Fanuc KAREL source: kt00536.KL

-- PROVISIONAL review KL for V770-1; original PC SHA256 9526b313598faa0eb3e1cc6d407e75327d356bfbb0ff6b673ecc31c0b60f6f1a
-- Incomplete behavior may be omitted. Consult companion uncertainty JSON. Do not deploy.
PROGRAM KT00536
%NOLOCKGROUP
-- UNRESOLVED_DECL P1 type=000199
-- UNRESOLVED_DECL P2 type=000101
-- UNRESOLVED_DECL OUT type=000106
BEGIN
  -- UNRESOLVED_PC offsets 5-39; opcodes 49,7E,49,60,7E,4A
  -- UNRESOLVED_PC offsets 44-48; opcodes 7F
END KT00536
